FUNCTION_BLOCK FB_CheckJack1_1
(*
	Description 	: Bloc fonction de gestion d'un module de mise sous vide
	Auteur		: DLA
	Date		: 26.03.2014
	Version		: 1.00

	Modifications :

*)
VAR_INPUT
	bJackGoOut	: BOOL;
	bJackIsOut	: BOOL;
	bResetErrors 	: BOOL;
	tTimeOut		: TIME			:= t#1s;
END_VAR
VAR_OUTPUT
	bJackError	: BOOL;
END_VAR
VAR
	T_Error		: TON;
	RSJackErr	: RS;
	bJackErr		: BOOL;
END_VAR

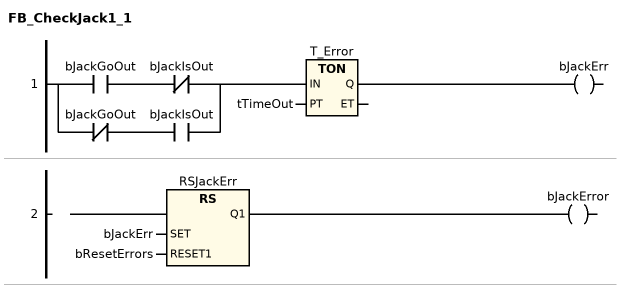
// NETWORK 1
T_Error(IN := bJackGoOut AND NOT bJackIsOut OR NOT bJackGoOut AND bJackIsOut, PT := tTimeOut); // TON
bJackErr := T_Error.Q;

// NETWORK 2
RSJackErr(SET := bJackErr, RESET1 := bResetErrors); // RS
bJackError := RSJackErr.Q1;

END_FUNCTION_BLOCK

(* stored: Version 1.1.0.1, ProductVersion 3.1.4022.12
   POU FB_CheckJack1_1: Id {3f876526-42f1-493a-af14-2445ce048729}, SpecialFunc None *)
